FUNCTION_BLOCK FB_Sequence
VAR_IN_OUT
	ServoAxis	:	AXIS_REF;			// Axises of two motors
	StepAxis	:	AXIS_REF;
END_VAR
VAR
	Slave		:	AXIS_REF;			// Slave and master axises
	Master		:	AXIS_REF;
	fbGearIn	:	MC_GearIn;			// Motion control function blocks
	fbMoveAbsolute	:	MC_MoveAbsolute;
	fbGearOut	:	MC_GearOut;
	fbResetServo 	: 			MC_Reset;
	fbResetStep 	: 			MC_Reset;
	fbPowerServo 	: 			MC_Power;
	xGearIn		:	BOOL;				// Coupling motors
	xGearOut	:	BOOL;				// Decoupling motors
    lrRatioNumerator   : LREAL:=1;
    uiRatioDenominator : UINT:=1;
	fbPowerStep	: 			MC_Power;
	xManualReset	 : 		BOOL; // Resetting program
	xPowerOn	:			BOOL; //Enabling power sources
	xExecute	:			BOOL; // Executing program
	eStateMc 	: 			E_MC ;		//instance of enum
	eStatePrevious	:		E_MC;
	xStepIsMaster		:		BOOL;
	xStepIsSlave	:		BOOL;
	lrPosition	: 			LREAL; 	//Target Position
	lrVelocity 	:			LREAL; 	// Setting Velocity
	lrRealPosition:			LREAL;	// real position
	xButton_NO1 	AT%I* : BOOL;
	xButton_NO2 	AT%I* : BOOL;
	xButton_NO3		AT%I* : BOOL;
	fTriggerStart			:	F_TRIG;
	fTriggerReset			:	F_TRIG;		// Falling triggers on 3 buttons
	fTriggerHome			:	F_TRIG;
	xStartSequence		:	BOOL;			// starting sequence
	xResetErrors		:	BOOL;			// Reseting errors
	xHomeMotors				:	BOOL;		// Homing motors
	tonTooLongInCase	:	TON;			// Ton timer counting time in each case
	xTooLongInCase		:	BOOL;		   // Too long in case
	sErrorLocalization	:	STRING(255);  // Moment when error occured
END_VAR

fTriggerStart(CLK:=xButton_NO2 , Q=>xStartSequence );		// Triggers on buttons
fTriggerReset(CLK:=xButton_NO1 , Q=>xResetErrors );
fTriggerHome(CLK:=xButton_NO3 , Q=>xHomeMotors );
lrRealPosition:=ServoAxis.NcToPlc.ActPos;
// Timer in each case
IF (eStateMc <> E_MC.Idle) AND (eStateMc <> E_MC.Error) AND (eStateMc <> E_MC.Execute) THEN
	IF eStateMc <> eStatePrevious THEN			// Comparing  current and previous values of enum
		tonTooLongInCase(IN := FALSE); 			// Reseting clock
		eStatePrevious := eStateMc; 			// timeout string
	END_IF

	tonTooLongInCase(IN := TRUE, PT :=T#15S);
	
	IF tonTooLongInCase.Q THEN
		eStateMc := E_MC.Error; 
		sErrorLocalization:='Timeout';
	END_IF
END_IF
// Case of program states
CASE eStateMc OF
	
	E_MC.Idle:									// Start of the program, homing
		IF xHomeMotors THEN
			xHomeMotors:=FALSE;
			eStateMc:=E_MC.RestartCall;
		END_IF
		
	E_MC.RestartCall:							// Calling reset of the errors
		xManualReset:=TRUE;							
		IF fbResetServo.Busy AND fbResetStep.Busy THEN
				eStateMc:=E_MC.RestartEffect;					
		ELSIF	fbResetServo.Error OR fbResetStep.Error THEN
			eStateMc:=E_MC.Error;
			sErrorLocalization:='Error when reseting motor errors(RestartCall)';
		END_IF
		
	E_MC.RestartEffect:						// Executing reset 
		xManualReset:=FALSE;
		IF fbResetServo.Done AND fbResetStep.Done THEN
			eStateMc:=E_MC.PowerCall;
		ELSIF	fbResetServo.Error OR fbResetStep.Error THEN
			eStateMc:=E_MC.Error;
			sErrorLocalization:='Error when reseting motor errors(RestartEffect)';
		END_IF
		
	E_MC.PowerCall:								// Calling power enable
		xPowerOn:=TRUE;
		IF fbPowerServo.Busy AND fbPowerStep.Busy THEN
				eStateMc:=E_MC.PowerEffect;
		ELSIF	fbPowerServo.Error OR fbPowerStep.Error THEN
			eStateMc:=E_MC.Error;
			sErrorLocalization:='Error when enabling motors power(PowerCall)';
		END_IF
		
	E_MC.PowerEffect:
		IF fbPowerServo.Status AND fbPowerStep.Status THEN
			eStateMc:=E_MC.HomingCallServo;
		ELSIF	fbPowerServo.Error OR fbPowerStep.Error THEN
			eStateMc:=E_MC.Error;
			sErrorLocalization:='Error when enabling motors power(PowerEffect)';
		END_IF
	
	E_MC.HomingCallServo:			// Homing servo motor
		Master:=ServoAxis;
		lrPosition:=0;
		lrVelocity:=100;
		xExecute:=TRUE;
		IF fbMoveAbsolute.Busy THEN
			eStateMc := E_MC.HomingEffectServo;
		END_IF
		IF fbMoveAbsolute.Error THEN
			// Going into error step, when error id is 1800 write information about it
			eStateMc:=E_MC.Error;
			IF ServoAxis.Status.ErrorID=16#00004650 THEN
				sErrorLocalization:=CONCAT(CONCAT('Error homing servo motor(HomingCallStep) ErrorID: ',UDINT_TO_STRING(ServoAxis.Status.ErrorID)),' Drive hardware not ready to operate');
			ELSE
				sErrorLocalization:='Error homing servo motor(HomingCallStep)';
			END_IF
		END_IF
		
	E_MC.HomingEffectServo:
		Master:=ServoAxis;
		xExecute:=FALSE;
		IF fbMoveAbsolute.Done THEN
			eStateMc:=E_MC.HomingCallStep;
		END_IF

		IF fbMoveAbsolute.Error THEN
			eStateMc:=E_MC.Error;
			IF ServoAxis.Status.ErrorID=16#00004650 THEN
				sErrorLocalization:=CONCAT(CONCAT('Error homing servo motor(HomingEffectServo) ErrorID: ',UDINT_TO_STRING(ServoAxis.Status.ErrorID)),' Drive hardware not ready to operate');
			ELSE
				sErrorLocalization:='Error homing servo motor(HomingEffectServo)';
			END_IF
		END_IF	

	E_MC.HomingCallStep:			// Homing Step motor
		Master:=StepAxis;
		lrPosition:=0;
		lrVelocity:=100;
		xExecute:=TRUE;
		IF fbMoveAbsolute.Busy THEN
			eStateMc := E_MC.HomingEffectStep;
		END_IF
		IF fbMoveAbsolute.Error THEN
			eStateMc:=E_MC.Error;
			IF StepAxis.Status.ErrorID=16#00004650 THEN
				sErrorLocalization:=CONCAT(CONCAT('Error homing servo motor(HomingCallStep) ErrorID: ',UDINT_TO_STRING(StepAxis.Status.ErrorID)),' Drive hardware not ready to operate');
			ELSE
				sErrorLocalization:='Error homing step motor(HomingCallStep)';
			END_IF			
		END_IF
		
	E_MC.HomingEffectStep:
		Master:=StepAxis;
		xExecute:=FALSE;
		IF fbMoveAbsolute.Done THEN
			eStateMc:=E_MC.Execute;
		END_IF

		IF fbMoveAbsolute.Error THEN
			eStateMc:=E_MC.Error;
			IF StepAxis.Status.ErrorID=16#00004650 THEN
				sErrorLocalization:=CONCAT(CONCAT('Error homing servo motor(HomingEffectStep) ErrorID: ',UDINT_TO_STRING(StepAxis.Status.ErrorID)),' Drive hardware not ready to operate');
			ELSE
				sErrorLocalization:='Error homing step motor(HomingEffectStep)';
			END_IF	
		END_IF		
	// Waiting for start button 
	E_MC.Execute:
		IF 	xStartSequence THEN
			xStartSequence:=FALSE;
			eStateMc:=E_MC.CoupleCallStepMaster;
		END_IF
		
	E_MC.CoupleCallStepMaster:					// Coupling Motors
		IF ServoAxis.Status.Coupled THEN
		eStateMc:=E_MC.MoveAbsCallStepMaster;
		END_IF
		Master := StepAxis;
		Slave  := ServoAxis;
		xGearIn:=TRUE;
		IF fbGearIn.Busy THEN
			eStateMc:=E_MC.CoupleEffectStepMaster;
		END_IF								
		IF fbGearIn.Error THEN
			eStateMc:=E_MC.Error;
			sErrorLocalization:='Error coupling motors(CoupleCallStepMaster)';
		END_IF
		
	E_MC.CoupleEffectStepMaster:
		IF fbGearIn.InGear  THEN
			eStateMc:=E_MC.MoveAbsCallStepMaster;
		ELSIF fbGearIn.Error THEN
			eStateMc:=E_MC.Error;
			sErrorLocalization:='Error coupling motors(CoupleEffectStepMaster)';
		END_IF	
	
	E_MC.MoveAbsCallStepMaster:				// move absolute for first coupling
		Master:=StepAxis;
		lrPosition:=720;
		lrVelocity:=100;
		xExecute:=TRUE;
		IF fbMoveAbsolute.Busy THEN
			eStateMc := E_MC.MoveAbsEffectStepMaster;
		END_IF
		IF fbMoveAbsolute.Error THEN
			eStateMc:=E_MC.Error;
			IF StepAxis.Status.ErrorID=16#00004650 THEN				// usunąc zera i zobaczyć czy działa
				sErrorLocalization:=CONCAT(CONCAT('Error in step motor movement(MoveAbsCallStepMaster) ErrorID: ',UDINT_TO_STRING(StepAxis.Status.ErrorID)),' Drive hardware not ready to operate');
			ELSIF ServoAxis.Status.ErrorID=16#00004650 THEN
				sErrorLocalization:=CONCAT(CONCAT('Error in servo motor movement(MoveAbsCallStepMaster) ErrorID: ',UDINT_TO_STRING(ServoAxis.Status.ErrorID)),' Drive hardware not ready to operate');
			ELSE
				sErrorLocalization:='Error in motors movement(MoveAbsCallStepMaster)';
			END_IF	
		END_IF
		
	E_MC.MoveAbsEffectStepMaster:
		Master:=StepAxis;
		xExecute:=FALSE;
		IF fbMoveAbsolute.Done THEN
			eStateMc:=E_MC.DecoupleCallStepMaster;
		END_IF

		IF fbMoveAbsolute.Error THEN
			eStateMc:=E_MC.Error;
			IF StepAxis.Status.ErrorID=16#00004650 THEN
				sErrorLocalization:=CONCAT(CONCAT('Error in step motor movement(MoveAbsEffectStepMaster) ErrorID: ',UDINT_TO_STRING(StepAxis.Status.ErrorID)),' Drive hardware not ready to operate');
			ELSIF ServoAxis.Status.ErrorID=16#00004650 THEN
				sErrorLocalization:=CONCAT(CONCAT('Error in servo motor movement(MoveAbsEffectStepMaster) ErrorID: ',UDINT_TO_STRING(ServoAxis.Status.ErrorID)),' Drive hardware not ready to operate');
			ELSE
				sErrorLocalization:='Error in motors movement(MoveAbsEffectStepMaster)';
			END_IF	
		END_IF	
	
	E_MC.DecoupleCallStepMaster:				// Decoupling motors
		xGearIn:=FALSE;
		xGearOut:=TRUE;
		Slave:=ServoAxis;
		IF fbGearOut.Busy THEN
			eStateMc:=E_MC.DecoupleEffectStepMaster;		
		ELSIF fbGearOut.Error THEN
			eStateMc:=E_MC.Error;
			sErrorLocalization:=CONCAT('Error decoupling motors	:	',TO_STRING(eStateMc));   // zmienić (attribute to string)
		END_IF	
		
	E_MC.DecoupleEffectStepMaster:
		xGearOut:=FALSE;
		Slave:=ServoAxis;
		IF fbGearOut.Done  THEN
			eStateMc:=E_MC.CoupleCallServoMaster;
		ELSIF fbGearOut.Error THEN
			eStateMc:=E_MC.Error;
			sErrorLocalization:='Error decoupling motors(DecoupleEffectStepMaster)';
		END_IF	
		
	E_MC.CoupleCallServoMaster:						// Second couple 
		IF StepAxis.Status.Coupled THEN
		eStateMc:=E_MC.MoveAbsCallServoMaster;
		END_IF
		
		Master := ServoAxis;
		Slave  := StepAxis;
		xGearIn:=TRUE;
		IF fbGearIn.Busy THEN
			eStateMc:=E_MC.CoupleEffectServoMaster;
		END_IF								
		IF fbGearIn.Error THEN
			eStateMc:=E_MC.Error;
			sErrorLocalization:='Error coupling motors(CoupleCallServoMaster)';
		END_IF	

	E_MC.CoupleEffectServoMaster:
		IF fbGearIn.InGear  THEN
			eStateMc:=E_MC.MoveAbsCallServoMaster;
		ELSIF fbGearIn.Error THEN
			eStateMc:=E_MC.Error;
			sErrorLocalization:='Error coupling motors(CoupleEffectServoMaster)';
		END_IF	

	E_MC.MoveAbsCallServoMaster:				// Move absolute for second couple
		Master := ServoAxis;
		lrPosition:=0;
		lrVelocity:=100;
		xExecute:=TRUE;
		IF fbMoveAbsolute.Busy THEN
			eStateMc := E_MC.MoveAbsEffectServoMaster;
		END_IF
		IF fbMoveAbsolute.Error THEN 
			eStateMc:=E_MC.Error;
			IF StepAxis.Status.ErrorID=16#00004650 THEN
				sErrorLocalization:=CONCAT(CONCAT('Error in step motor movement(MoveAbsCallServoMaster) ErrorID: ',UDINT_TO_STRING(StepAxis.Status.ErrorID)),' Drive hardware not ready to operate');
			ELSIF ServoAxis.Status.ErrorID=16#00004650 THEN
				sErrorLocalization:=CONCAT(CONCAT('Error in servo motor movement(MoveAbsCallServoMaster) ErrorID: ',UDINT_TO_STRING(ServoAxis.Status.ErrorID)),' Drive hardware not ready to operate');
			ELSE
				sErrorLocalization:='Error in motors movement(MoveAbsCallServoMaster)';
			END_IF	
		END_IF
	
	E_MC.MoveAbsEffectServoMaster:
		Master:=ServoAxis;
		xExecute:=FALSE;
		IF fbMoveAbsolute.Done THEN
			eStateMc:=E_MC.DecoupleCallServoMaster;
		END_IF
		
		IF fbMoveAbsolute.Error THEN
			eStateMc:=E_MC.Error;
			IF StepAxis.Status.ErrorID=16#00004650 THEN
				sErrorLocalization:=CONCAT(CONCAT('Error in step motor movement(MoveAbsEffectServoMaster) ErrorID: ',UDINT_TO_STRING(StepAxis.Status.ErrorID)),' Drive hardware not ready to operate');
			ELSIF ServoAxis.Status.ErrorID=16#00004650 THEN
				sErrorLocalization:=CONCAT(CONCAT('Error in servo motor movement(MoveAbsEffectServoMaster) ErrorID: ',UDINT_TO_STRING(ServoAxis.Status.ErrorID)),' Drive hardware not ready to operate');
			ELSE
				sErrorLocalization:='Error in motors movement(MoveAbsEffectServoMaster)';
			END_IF	
		END_IF					
	
	E_MC.DecoupleCallServoMaster:				// Decoupling
		xGearIn:=FALSE;
		xGearOut:=TRUE;
		Slave:=StepAxis;
		IF fbGearOut.Busy THEN
			eStateMc:=E_MC.DecoupleEffectServoMaster;		
		ELSIF fbGearOut.Error THEN
			eStateMc:=E_MC.Error;
			sErrorLocalization:='Error decoupling motors(DecoupleCallServoMaster)';
		END_IF	
		
		
	E_MC.DecoupleEffectServoMaster:
		xGearOut:=FALSE;
		Slave:=StepAxis;
		IF fbGearOut.Done  THEN
			eStateMc:=E_MC.Idle;
		ELSIF fbGearOut.Error THEN
			eStateMc:=E_MC.Error;
			sErrorLocalization:='Error decoupling motors(DecoupleEffectServoMaster)';
		END_IF		
	
		
	// Cases for when error occurs 	
		
	E_MC.DecoupleCallOnReset:							// Decoupling after reset
		IF StepAxis.Status.Coupled THEN
			Slave:=StepAxis;
		ELSIF ServoAxis.Status.Coupled THEN
			Slave:=ServoAxis;
		END_IF
		xGearIn:=FALSE;
		xGearOut:=TRUE;
		IF fbGearOut.Busy THEN
			eStateMc:=E_MC.DecoupleEffectOnReset;		
		ELSIF fbGearOut.Error THEN
			eStateMc:=E_MC.Error;
			sErrorLocalization:='Error decoupling motors(DecoupleCallOnReset)';
		END_IF	
	
	E_MC.DecoupleEffectOnReset:	
		IF StepAxis.Status.Coupled THEN
			Slave:=StepAxis;
		ELSIF ServoAxis.Status.Coupled THEN
			Slave:=ServoAxis;
		END_IF
		xGearOut:=FALSE;
		Slave:=StepAxis;
		IF fbGearOut.Done  THEN
			eStateMc:=E_MC.RestartCallOnReset;
		ELSIF fbGearOut.Error THEN
			eStateMc:=E_MC.Error;
			sErrorLocalization:='Error decoupling motors(DecoupleEffectOnReset)';
		END_IF		
		
	E_MC.RestartCallOnReset:									// Reseting errors after reset 
		xManualReset:=TRUE;							
		IF fbResetServo.Busy AND fbResetStep.Busy THEN
				eStateMc:=E_MC.RestartEffectOnReset;					
		ELSIF	fbResetServo.Error OR fbResetStep.Error THEN
			eStateMc:=E_MC.Error;
			sErrorLocalization:='Error when reseting motor errors(RestartCallOnReset)';
		END_IF
		
	E_MC.RestartEffectOnReset:	
		xManualReset:=FALSE;
		IF fbResetServo.Done AND fbResetStep.Done THEN
			eStateMc:=E_MC.Idle;
		ELSIF	fbResetServo.Error OR fbResetStep.Error THEN
			eStateMc:=E_MC.Error;
			sErrorLocalization:='Error when reseting motor errors(RestartEffectOnReset)';
		END_IF
		
	E_MC.Error:									// Error case, turning power off and going to next case
		xPowerOn:=FALSE;
		IF xResetErrors THEN
			xResetErrors:=FALSE;
			sErrorLocalization:='';
			IF StepAxis.Status.Coupled OR ServoAxis.Status.Coupled THEN
				eStateMc := E_MC.DecoupleCallOnReset;
			ELSE
				eStateMc := E_MC.RestartCallOnReset;
			END_IF	
		END_IF
END_CASE


//SERVO MOTOR
fbResetServo(				//Reseting motor // Reset1 -> ResetServoMotor
	Axis:= ServoAxis, 
	Execute:= xManualReset, 
	Done=> , 
	Busy=> , 
	Error=> , 
	ErrorID=> );
	
fbPowerServo(				// Turning power on
	Axis:= ServoAxis, 
	Enable:= xPowerOn, 
	Enable_Positive:= xPowerOn, 
	Enable_Negative:= xPowerOn, 
	Override:= 100, 
	BufferMode:= , 
	Options:= , 
	Status=> , 
	Busy=> , 
	Error=> , 
	ErrorID=> );
	
	
//STEP MOTOR
fbResetStep(				//Reseting motor
	Axis:= StepAxis, 
	Execute:= xManualReset, 
	Done=> , 
	Busy=> , 
	Error=> , 
	ErrorID=> );
	
fbPowerStep(				// Turning power on
	Axis:= StepAxis, 
	Enable:= xPowerOn, 
	Enable_Positive:= xPowerOn, 
	Enable_Negative:= xPowerOn, 
	Override:= 100, 
	BufferMode:= , 
	Options:= , 
	Status=> , 
	Busy=> , 
	Error=> , 
	ErrorID=> );
	
	
fbMoveAbsolute(			// Executing program
	Axis:= Master, 
	Execute:= xExecute, 
	Position:=lrPosition, 
	Velocity:= lrVelocity, 
	Acceleration:= , 
	Deceleration:= , 
	Jerk:= , 
	BufferMode:= , 
	Options:= , 
	Done=> , 
	Busy=> , 
	Active=> , 
	CommandAborted=> , 
	Error=> , 
	ErrorID=> );
fbGearIn(
		Master:=Master , 
		Slave:=Slave , 
		Execute:=xGearIn , 
		RatioNumerator:=lrRatioNumerator , 
		RatioDenominator:= uiRatioDenominator, 
		Acceleration:= , 
		Deceleration:= , 
		Jerk:= , 
		BufferMode:= , 
		Options:= , 
		InGear=> , 
		Busy=> , 
		Active=> , 
		CommandAborted=> , 
		Error=> , 
		ErrorID=> );
	
fbGearOut(
		Slave:= Slave, 
		Execute:=xGearOut , 
		Options:= , 
		Done=> , 
		Busy=> , 
		Error=> , 
		ErrorID=> );

END_FUNCTION_BLOCK

(* stored: Version 1.1.0.1, ProductVersion 3.1.4024.13
   POU FB_Sequence: Id {78c0308a-89d8-46d6-9315-ac5ef803a704}, SpecialFunc None *)
